PROGRAM OkToRun
VAR

	alarmTimeout: TON := (PT := TIME#11S0MS);
	
END_VAR

alarmTimeout();

//HARD CODED UPPER AND LOWER LIMITS
IF GVL.Temp > 50 THEN
		GVL.bCriticalAlarm:=TRUE;
		IO_VARS.ENABLE:=FALSE;
		GVL.sAlarmText:='Critical High Temp Alarm';
	END_IF
IF GVL.Temp < 0 THEN
	GVL.bCriticalAlarm:=TRUE;
	IO_VARS.ENABLE:=FALSE;
	GVL.sAlarmText:='Critical Low Temp Alarm';
END_IF



//If not in manual mode
IF GVL.manualMode=FALSE THEN
	
	//If running
	IF GVL.iState=1 THEN

	
		//Temperature Alarm Logic for STEP MODE
		IF GVL.TempStepmode THEN
			IF GVL.iState=1 AND GVL.Temp > (GVL.TempAlarmHigh) THEN
				GVL.bCriticalAlarm:=TRUE;
				GVL.sAlarmText:='High Temp Alarm';
			END_IF
			IF GVL.iState=1 AND GVL.Temp < (GVL.TempAlarmLow) THEN
				GVL.bCriticalAlarm:=TRUE;
				GVL.sAlarmText:='Low Temp Alarm';
			END_IF
		END_IF
		
		//Temperature alarm logic for RAMP MODE
		IF GVL.TempStepmode=FALSE THEN
			IF GVL.iState=1 AND GVL.Temp > (GVL.TempSetpoint+GVL.TempAlarmHigh) THEN
				GVL.bCriticalAlarm:=TRUE;
				GVL.sAlarmText:='High Temp Alarm';
			END_IF
			IF GVL.iState=1 AND GVL.Temp < (GVL.TempSetpoint-GVL.TempAlarmLow) THEN
				GVL.bCriticalAlarm:=TRUE;
				GVL.sAlarmText:='Low Temp Alarm';
			END_IF
		END_IF
		
		//Schedule Alarms
		//If the user deletes the current program or changes the schedule in an incorrect way, 
		//Tell them they messed up
		//This could also happen if there are database errors
		IF fbGetCurrentScheduleLine.sSeverity="No Error" AND fbGetCurrentScheduleLine.iLines=0 THEN
			alarmTimeout.IN:=TRUE;
			IF alarmTimeout.Q=TRUE THEN
				GVL.sAlarmText:='Error getting current program. Check schedule and programs';
				GVL.bCriticalAlarm:=TRUE;
				alarmTimeout.IN:=FALSE;
				
			END_IF
				
		ELSE

			alarmTimeout.IN:=FALSE;
			
		END_IF
		//Temperature sensor alarm
		IF ABS((GVL.Temp-GVL.Temp2)*100/GVL.Temp)>GVL.TempCalibrationLimit THEN
				GVL.sAlarmText:='Temperature Sensor Error.';
				GVL.bCriticalAlarm:=TRUE;
		END_IF
		
		//Humidity sensor alarm
		IF ABS((GVL.Humidity-GVL.Humidity2)*100/GVL.Humidity)>GVL.HumCalibrationLimit THEN
				GVL.sAlarmText:='Humidity Sensor Error.';
				GVL.bCriticalAlarm:=TRUE;
		END_IF
		

	END_IF
	
	

END_IF	

//OK TO RUN IF THERE ARE NO ERRORS
IF GVL.bCriticalAlarm=FALSE AND GVL.HMIPowerButton=TRUE THEN
	GVL.okToRun:=TRUE;
	GVL.sAlarmText:='Running No Alarm';
	IO_VARS.ENABLE:=TRUE;
ELSIF GVL.bCriticalAlarm=FALSE AND GVL.HMIPowerButton=FALSE AND IO_VARS.ENABLE=FALSE THEN
	GVL.sAlarmText:='Not Running No Alarm';
ELSE
	GVL.okToRun:=FALSE;
	IF GVL.manualMode=FALSE THEN
		IO_VARS.ENABLE:=FALSE;
	END_IF
	
	GVL.HMIPowerButton:=FALSE;
END_IF

END_PROGRAM

(* stored: Version 1.1.0.1, ProductVersion 3.1.4022.18
   POU OkToRun: Id {31a4ced2-eb7b-4495-8b26-88a3f28b5673}, SpecialFunc None *)
